{attribute 'qualified_only'}
{attribute 'strict'}
{attribute 'to_string'}
TYPE eCommunicationState :
(
	DISCONNECTED,
    CONNECTING,
    CONNECTED,
    DISCONNECTING,
    ERROR
);
END_TYPE

(* stored: Version 1.1.0.1, ProductVersion 3.1.4026.18
   DUT eCommunicationState: Id {454aae8e-62f1-43e1-a34f-404d20f80024} *)
